PROGRAM Ext_SP_Gen
VAR
	bMstrExtSP			: BOOL;
	ExtSP_Enable		: MC_ExtSetPointGenEnable;
	ExtSP_Disable		: MC_ExtSetPointGenDisable;	

	lrPosCmd			: LREAL;
	lrVeloCmd			: LREAL;
	lrAccelCmd			: LREAL;

	rDeg				: REAL;
	rDegStep			: REAL := 0.1;
	lrSinWave			: LREAL;
	rSinAmp				: REAL := 30.0;
	
	bSinGen				: BOOL;
	bAddSin				: BOOL;

	diDir: DINT := 1;
	
	lrPosInput: LREAL;
END_VAR

IF bSinGen THEN
	rDeg:=rDeg+rDegStep;
	IF rDeg >= 360.0 THEN
		rDeg:=0.0;
	END_IF
END_IF

lrSinWave:=rSinAmp*SIN(rDeg*3.14159/180.0);	// SIN function uses radian input

IF bAddSin THEN
	lrPosCmd:=lrPosInput+lrSinWave;
ELSE
	lrPosCmd:=lrPosInput;
END_IF

MC_ExtSetPointGenFeed(
	lrPosCmd,
	lrVeloCmd,
	lrAccelCmd,
	diDir,
	stAxis3);

ExtSP_Enable(
	Axis:= stAxis3, 
	Execute:= bMstrExtSP, 
	Position:= , 
	PositionType:= POSITIONTYPE_ABSOLUTE, 
	Done=> , 
	Busy=> , 
	Error=> , 
	ErrorID=> , 
	Enabled=> );
	
ExtSP_Disable(
	Axis:= stAxis3, 
	Execute:= NOT(bMstrExtSP), 
	Done=> , 
	Busy=> , 
	Error=> , 
	ErrorID=> , 
	Enabled=> );

END_PROGRAM

(* stored: Version 1.1.0.1, ProductVersion 3.1.4024.11
   POU Ext_SP_Gen: Id {b7780f01-6728-483a-8a18-a828f1046393}, SpecialFunc None *)
